// TIA Portal V18 export
DATA_BLOCK "MainDB"   // DB30
{ S7_Optimized_Access := 'TRUE' }
VERSION : 0.1
// stored: AutoNumber true, DBAccessibleFromOPCUA true, IsOnlyStoredInLoadMemory false, IsRetainMemResEnabled false, IsWriteProtectedInAS false, MemoryReserve 100
   VAR
      Monitor : Bool;
      Step0M : Bool;
      Step0 : Bool;
      Step10 : Bool;
      Step20 : Bool;
      Step30 : Bool;
      Step40 : Bool;
      Step50 : Bool;
      Step0_10 : Bool;
      Step10_20 : Bool;
      Step20_30 : Bool;
      Step30_40 : Bool;
      Step40_50 : Bool;
      Step50_10 : Bool;
      ESTOPEdgeMemory : Bool;
      ESTOPEdge : Bool;
      AllAxisFaultRelease : Bool;
      Step0MConfig : Bool;
   END_VAR
BEGIN
END_DATA_BLOCK
